// TIA Portal project "MES_DB_ALOCATION" (V15.1)

(* hardware
DEVICE "S71500/ET200MP station_1"  S7-1500 station
   slot 0: "Rail_0"  Rack  6ES7 590-1***0-0AA0
   slot 1: "PLC_1"  CPU 1513F-1 PN  6ES7 513-1FL02-0AB0  V2.6
      slot 3: "CPU display_1"  6ES7591-1AA00-0AA0
*)

// ===== PLC "PLC_1"  CPU 1513F-1 PN =====

DATA_BLOCK "Main_Safety_RTG1_DB"   // DB1, F_DB
{ S7_Optimized_Access := 'TRUE' }
NAME : FUSI
VERSION : 0.1
// stored: InstanceOfName Main_Safety_RTG1
"Main_Safety_RTG1"
BEGIN
END_DATA_BLOCK

DATA_BLOCK "MES_DB1"   // DB2
{ S7_Optimized_Access := 'FALSE' }
VERSION : 0.1
   VAR
      LiveCheck : Byte;
      JIT_status : Byte;   // ListenerStarting:0;Listening:1;ReadyForCycle:2;CycleRejected:3
      PLC_status : Byte;   // InitiatorStarting:0;InitiatorStarted:1;CycleCompleted:2;FixtureReady:3
      JobNr : Array[0..9] of Char;
      CallOffDateTime : Array[0..15] of Char;
      VehicleNo : Array[0..12] of Char;
      RearWindowType : String[18];
      Model : Byte;
   END_VAR
BEGIN
END_DATA_BLOCK

DATA_BLOCK "Default_SupervisionDB"   // DB3
{ S7_Optimized_Access := 'TRUE' }
VERSION : 0.1
// stored: InstanceOfName Default_SupervisionFB
"Default_SupervisionFB"
BEGIN
END_DATA_BLOCK

DATA_BLOCK "MES_DB3"   // DB4
{ S7_Optimized_Access := 'FALSE' }
VERSION : 0.1
   VAR
      LiveCheck : Byte;
      JIT_status : Byte;   // ListenerStarting:0;Listening:1;ReadyForCycle:2;CycleRejected:3
      PLC_status : Byte;   // InitiatorStarting:0;InitiatorStarted:1;CycleCompleted:2;FixtureReady:3
      JobNr : Array[0..9] of Char;
      VehicleNo : Array[0..12] of Char;
      RearWindowType : String[18];
      GlassID : Array[0..9] of Char;
      flag4 : Bool;
   END_VAR
BEGIN
END_DATA_BLOCK

DATA_BLOCK "MES_DB2"   // DB5
{ S7_Optimized_Access := 'FALSE' }
VERSION : 0.1
   VAR
      LiveCheck : Byte;
      JIT_status : Byte;   // ListenerStarting:0;Listening:1;ReadyForCycle:2;CycleRejected:3
      PLC_status : Byte;   // InitiatorStarting:0;InitiatorStarted:1;CycleCompleted:2;FixtureReady:3
      JobNr : Array[0..9] of Char;
      VehicleNo : Array[0..12] of Char;
      RearWindowType : String[18];
   END_VAR
BEGIN
END_DATA_BLOCK

FUNCTION_BLOCK "Main_Safety_RTG1"   // FB1, F_FBD
{ S7_Optimized_Access := 'TRUE' }
VERSION : 0.1
BEGIN
END_FUNCTION_BLOCK

FUNCTION_BLOCK "Default_SupervisionFB"   // FB2, ProDiag
{ S7_Optimized_Access := 'TRUE' }
   VAR
      PC_Flags : PC_Flags_V2;
      State : SV_FB_State_V2;
   END_VAR
   VAR_TEMP
      t_TempSvStateUDT : SV_State_V2;
      t_TempAlarmInstance : <type 200004f>;
      t_TempAsocValue1 : Variant;
      t_TempAsocValue2 : Variant;
      t_TempAsocValue3 : Variant;
   END_VAR
BEGIN
END_FUNCTION_BLOCK

ORGANIZATION_BLOCK "Main"   // OB1, LAD, ProgramCycle
TITLE = "Main Program Sweep (Cycle)"
{ S7_Optimized_Access := 'TRUE' }
VERSION : 0.1
   VAR_INPUT
      Initial_Call : Bool;   // Initial call of this OB
      Remanence : Bool;   // =True, if remanent data are available
   END_VAR
BEGIN
END_ORGANIZATION_BLOCK

ORGANIZATION_BLOCK "ProDiagOB"   // OB250, ProDiag_OB, ProgramCycle
TITLE = "Main Program Sweep (Cycle)"
{ S7_Optimized_Access := 'TRUE' }
VERSION : 0.1
   VAR_INPUT
      Initial_Call : Bool;   // Initial call of this OB
      Remanence : Bool;   // =True, if remanent data are available
   END_VAR
BEGIN

REGION Network 1
   CALL "Default_SupervisionFB", "Default_SupervisionDB";
END_REGION
END_ORGANIZATION_BLOCK